PROGRAM Instanziierne
VAR
	BasisSkill			:SkillBasisGeruest;
	SkillTest			:SkillNeu;
END_VAR

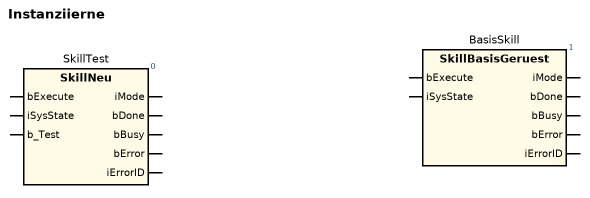
SkillTest(); // SkillNeu
BasisSkill(); // SkillBasisGeruest

END_PROGRAM

(* stored: Version 1.1.0.1
   POU Instanziierne: Id {7f1fc299-89d9-48e1-bf2a-216988907bbf}, SpecialFunc None *)
